TYPE ST_Motor :
STRUCT
	sDesc			:STRING;   //  Description or name of equipment
	rSpeed			:REAL;	   //  Speed of motor
	rPosition		:REAL;	   // Position of motor
END_STRUCT
END_TYPE

(* stored: Version 1.1.0.1, ProductVersion 3.1.4024.12
   DUT ST_Motor: Id {3108c199-6a05-4188-b458-a71e1fad5edc} *)
